(* PLC project Senza_nome, Sconosciuto Senza_nome 1 *)
(* stored: creationDateTime 2021-04-12T13:03:08, modificationDateTime 2021-04-12T14:28:47 *)

PROGRAM carrello
  VAR_INPUT
    start_button : BOOL;  (* Pulsante di avvio *)
  END_VAR
  VAR_EXTERNAL
    go_right : BOOL;  (* Sposta il carrello verso destra *)
    go_left : BOOL;  (* Sposta il carrello verso sinistra *)
    load : BOOL;  (* Ribalta il serbatoio per caricare il carrello *)
    fd : BOOL;  (* Finecorsa dx *)
    fs : BOOL;  (* Finecorsa sx *)
    fr : BOOL;  (* Finecorsa serbatoio *)
  END_VAR
  VAR  (* added by the conversion: wires and edge detectors of the diagram *)
    R_TRIG1 : R_TRIG;
  END_VAR

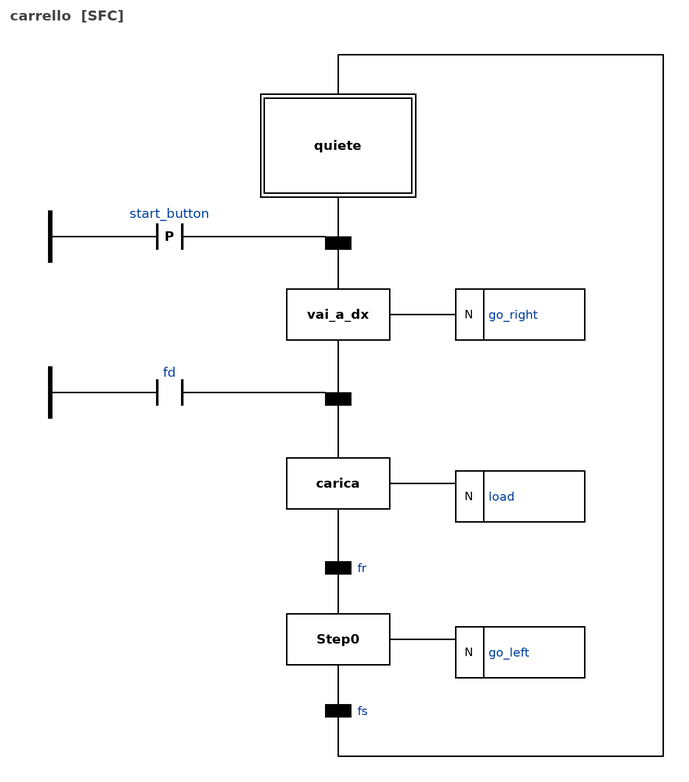
INITIAL_STEP quiete:
  COMPUTE_FUNCTION_BLOCKS(S);
END_STEP
TRANSITION FROM quiete TO vai_a_dx
  := R_TRIG1.Q;
END_TRANSITION
STEP vai_a_dx:
  go_right(N);
END_STEP
TRANSITION FROM vai_a_dx TO carica
  := fd;
END_TRANSITION
STEP carica:
  load(N);
END_STEP
TRANSITION FROM carica TO Step0
  := fr;
END_TRANSITION
STEP Step0:
  go_left(N);
END_STEP
TRANSITION FROM Step0 TO quiete
  := fs;
END_TRANSITION
ACTION COMPUTE_FUNCTION_BLOCKS:  (* blocks drawn on the SFC sheet *)
  R_TRIG1(CLK := start_button);
END_ACTION
END_PROGRAM

PROGRAM simulazione_carrello
  VAR
    dummy1 : BOOL := 0;  (* dummy timer *)
    dummy2 : BOOL := 0;  (* dummy timer *)
    dummy3 : BOOL := 0;  (* dummy timer *)
  END_VAR
  VAR_EXTERNAL
    go_right : BOOL;
    go_left : BOOL;
    load : BOOL;
    fd : BOOL;
    fs : BOOL;
    fr : BOOL;
  END_VAR

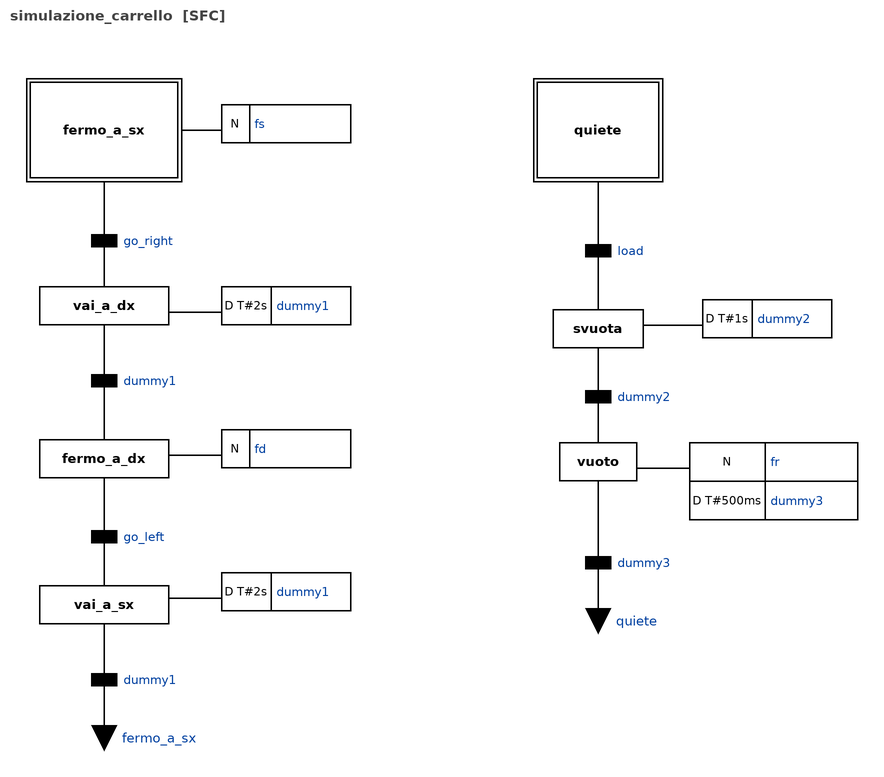
INITIAL_STEP fermo_a_sx:
  fs(N);
END_STEP
TRANSITION FROM fermo_a_sx TO vai_a_dx
  := go_right;
END_TRANSITION
INITIAL_STEP quiete:
END_STEP
TRANSITION FROM quiete TO svuota
  := load;
END_TRANSITION
STEP vai_a_dx:
  dummy1(D, T#2s);
END_STEP
TRANSITION FROM vai_a_dx TO fermo_a_dx
  := dummy1;
END_TRANSITION
STEP svuota:
  dummy2(D, T#1s);
END_STEP
TRANSITION FROM svuota TO vuoto
  := dummy2;
END_TRANSITION
STEP fermo_a_dx:
  fd(N);
END_STEP
TRANSITION FROM fermo_a_dx TO vai_a_sx
  := go_left;
END_TRANSITION
STEP vuoto:
  fr(N);
  dummy3(D, T#500ms);
END_STEP
TRANSITION FROM vuoto TO quiete
  := dummy3;
END_TRANSITION
STEP vai_a_sx:
  dummy1(D, T#2s);
END_STEP
TRANSITION FROM vai_a_sx TO fermo_a_sx
  := dummy1;
END_TRANSITION
END_PROGRAM

CONFIGURATION Config0
  RESOURCE Res0 ON PLC
    VAR_GLOBAL
      go_right : BOOL;
      go_left : BOOL;
      load : BOOL;
      fs : BOOL;
      fd : BOOL;
      fr : BOOL;
    END_VAR
    TASK task0(INTERVAL := T#20ms, PRIORITY := 0);
    TASK task1(INTERVAL := T#100ms, PRIORITY := 1);
    PROGRAM controllo WITH task0 : carrello;
    PROGRAM simulazione WITH task1 : simulazione_carrello;
  END_RESOURCE
END_CONFIGURATION
